// TIA Portal project "Set y Reset FI" (V17)

(* hardware
DEVICE "S7-1200 station_1"  S7-1200 Station
   slot 0: "Rack_0"  S7-1200 Rack  Rack  V1.0
   slot 1: "PLC_1"  CPU 1212C AC/DC/Rly  6ES7 212-1BE40-0XB0  V4.5
*)

// ===== PLC "PLC_1"  CPU 1212C AC/DC/Rly =====

VAR_GLOBAL   // PLC tag table "Default tag table"
   "Arranque" AT %I0.0 : Bool;
   "Paro" AT %I0.1 : Bool;
   "M" AT %M0.0 : Bool;
   "Sensor 1" AT %I0.2 : Bool;
   "Sensor 2" AT %I0.3 : Bool;
   "Paro de Emergencia" AT %I0.4 : Bool;
   "Led Verde" AT %Q0.0 : Bool;
   "Led Rojo" AT %Q0.1 : Bool;
   "Motor" AT %Q0.2 : Bool;
END_VAR

FUNCTION "MHJ-PLC-Lab-Function-S71200" : Void   // FC9000, SCL
{ S7_Optimized_Access := 'TRUE' }
VERSION : 0.1
   VAR_TEMP
      rdTimeReturn : Int;
      outputTime : DTL;
      SyncVal : Byte;
      forVal : Int;
      forVal_2 : Int;
      Value : Byte;
   END_VAR
   VAR CONSTANT
      CompVal : Byte := 16#34;
      Value_01 : Byte := 16#11;
      Value_01_DW : DWord := 16#A165_D992;
      Value_02_DW : DWord := 16#58BE_4401;
   END_VAR
BEGIN

   #Value:=PEEK(area := 16#82,
        dbNumber := 0,
        byteOffset := 511);
   #Value := #Value + 1;

   POKE(area := 16#82,
        dbNumber := 0,
        byteOffset := 511,
        value := #Value);

   POKE(area:=16#81,
        dbNumber:=0,
        byteOffset:=1016,
        value:=#Value_01_DW);
   POKE(area := 16#81,
        dbNumber := 0,
        byteOffset := 1020,
        value := #Value_02_DW);

   POKE(area := 16#81,
        dbNumber := 0,
        byteOffset := 511,
        value := B#16#00);

   FOR #forVal := 0 TO 120 DO
       FOR #forVal_2:=0 TO 10 DO
           #rdTimeReturn:=RD_SYS_T(#outputTime);
           #rdTimeReturn := WR_SYS_T(#outputTime);
           #rdTimeReturn := RD_SYS_T(#outputTime);
           #rdTimeReturn := WR_SYS_T(#outputTime);
       END_FOR;
       #SyncVal:= PEEK(area := 16#81,
                      dbNumber := 0,
                      byteOffset := 511);
       IF #SyncVal = #CompVal THEN
          GOTO M_1;
       END_IF;
   END_FOR;
   RETURN;

   M_1:
   POKE(area := 16#81,
        dbNumber := 0,
        byteOffset := 511,
        value := B#16#0);
END_FUNCTION

ORGANIZATION_BLOCK "Main"   // OB1, LAD, ProgramCycle
TITLE = "Main Program Sweep (Cycle)"
{ S7_Optimized_Access := 'TRUE' }
VERSION : 0.1
   VAR_INPUT
      Initial_Call : Bool;   // Initial call of this OB
      Remanence : Bool;   // =True, if remanent data are available
   END_VAR
BEGIN

REGION Network 1: Conexión Factory IO
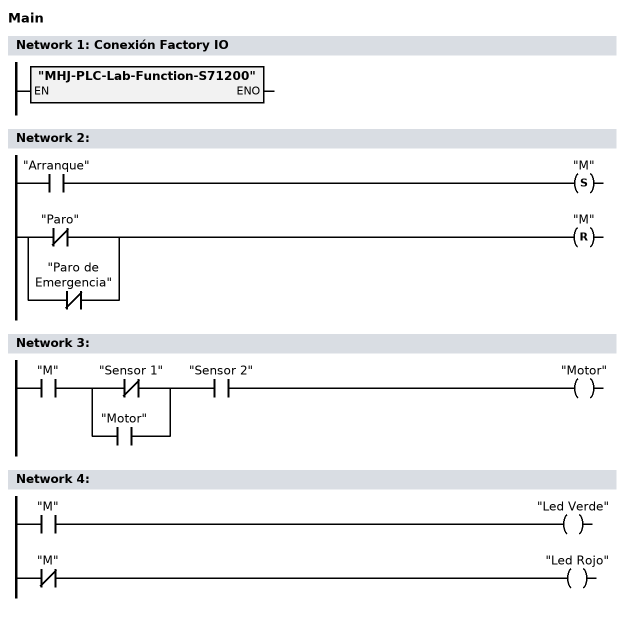
   RUNG wire#powerrail
      "MHJ-PLC-Lab-Function-S71200"()
   END_RUNG
   // the same network as SCL:
   "MHJ-PLC-Lab-Function-S71200"();
END_REGION

REGION Network 2
   RUNG wire#powerrail
      Contact( "Arranque" )
      S_Coil( "M" )
   END_RUNG
   RUNG wire#powerrail
      I_Contact( "Paro" )
      wire#w1
      R_Coil( "M" )
   END_RUNG
   RUNG wire#powerrail
      I_Contact( "Paro de Emergencia" )
   END_RUNG wire#w1
   // the same network as SCL:
   IF "Arranque" THEN "M" := TRUE; END_IF;
   IF NOT "Paro" OR NOT "Paro de Emergencia" THEN "M" := FALSE; END_IF;
END_REGION

REGION Network 3
   RUNG wire#powerrail
      Contact( "M" )
      wire#w1
      I_Contact( "Sensor 1" )
      wire#w2
      Contact( "Sensor 2" )
      Coil( "Motor" )
   END_RUNG
   RUNG wire#w1
      Contact( "Motor" )
   END_RUNG wire#w2
   // the same network as SCL:
   "Motor" := "M" AND (NOT "Sensor 1" OR "Motor") AND "Sensor 2";
END_REGION

REGION Network 4
   RUNG wire#powerrail
      Contact( "M" )
      Coil( "Led Verde" )
   END_RUNG
   RUNG wire#powerrail
      I_Contact( "M" )
      Coil( "Led Rojo" )
   END_RUNG
   // the same network as SCL:
   "Led Verde" := "M";
   "Led Rojo" := NOT "M";
END_REGION
END_ORGANIZATION_BLOCK